FUNCTION_BLOCK FB_StatePMPSLimits_Test EXTENDS MotorTestSuite
(*
    Tests for FB_StatePMPSLimits

    This function block ensures that:
    - When not at our goal state, we cannot move away from our goal state
    - When at our goal state, we must stay within the state bounds
    - When at our goal state, we still obey other constraints like limit switches
*)
VAR
    stMotionStage: ST_MotionStage;
    fbMotionStage: FB_MotionStage;
    astPositionState: ARRAY[1..GeneralConstants.MAX_STATES] OF ST_PositionState;
    fbInternal1: FB_PositionStateInternal;
    fbInternal2: FB_PositionStateInternal;
    nInvalidState: UINT := 2;
    nGoalState: UINT := 4;
    nNotUpdatedState: UINT := 6;

    bInit: BOOL;
    nTestCounter: UINT;
    bOneTestDone: BOOL;
    fTestStartPos: LREAL;
    tonTimer: TON;
    bStatesReady: BOOL;
END_VAR


astPositionState[nGoalState].fPosition := 10;
astPositionState[nGoalState].fDelta := 1;
SetGoodState(astPositionState[nGoalState]);
astPositionState[nInvalidState].fPosition := 20;
astPositionState[nInvalidState].fDelta := 1;
astPositionState[nNotUpdatedState].fPosition := 20;
astPositionState[nNotUpdatedState].fDelta := 1;
SetGoodState(astPositionState[nNotUpdatedState]);
fbInternal1(
    stMotionStage:=stMotionStage,
    stPositionState:=astPositionState[nGoalState],
);
fbInternal2(
    stMotionStage:=stMotionStage,
    stPositionState:=astPositionState[nInvalidState],
);
fbMotionStage(stMotionStage:=stMotionStage);
bStatesReady:=astPositionState[nGoalState].bUpdated AND astPositionState[nInvalidState].bUpdated;

IF bStatesReady AND nTestCounter = 0 THEN
    // Don't run any tests until the states are ready
    nTestCounter := 1;
END_IF

TestInvalid(1);
TestNotUpdated(2);
TestBelow(3);
TestAbove(4);
TestAt(5);
TestDisabled(6);
TestLimits(7);

IF bOneTestDone THEN
    bOneTestDone := FALSE;
    nTestCounter := nTestCounter + 1;
    tonTimer(IN:=FALSE);
END_IF
// Use this timer to time out any tests that stall
tonTimer(
    IN:=bStatesReady,
    PT:=T#5s,
);

METHOD TestAbove
VAR_INPUT
    nTestID: UINT;
END_VAR
VAR_INST
    fbStateLimits: FB_StatePMPSLimits;
    fbFFHWO: FB_HardwareFFOutput := (bAutoReset := TRUE);
    fbMove: FB_TestHelperSetAndMove;

    bInit: BOOL;
END_VAR

TEST('TestAbove');
IF nTestCounter <> nTestID THEN
    RETURN;
END_IF

SetEnablesPMPS(stMotionStage);

// Set position to be above the goal's range
fbMove(
    stMotionStage:=stMotionStage,
    bExecute:=bInit,
    fStartPosition:=astPositionState[nGoalState].fPosition + 100 * astPositionState[nGoalState].fDelta,
    fGoalPosition:=astPositionState[nGoalState].fPosition + 100 * astPositionState[nGoalState].fDelta,
    fVelocity:=1,
    bHWEnable:=FALSE,
);
bInit := TRUE;
// Run our FB
fbStateLimits(
    stMotionStage:=stMotionStage,
    astPositionState:=astPositionState,
    fbFFHWO:=fbFFHWO,
    bEnable:=TRUE,
    nGoalStateIndex:=nGoalState,
);
fbFFHWO.EvaluateOutput();
// If we've set the position OR ran out of time to set the position, check the asserts
IF tonTimer.Q OR fbMove.bSetDone THEN
    AssertFalse(
        tonTimer.Q,
        'Timeout in test',
    );
    AssertEquals_LREAL(
        Expected:=fbMove.fStartPosition,
        Actual:=fbMove.fActPosition,
        Delta:=0.0001,
        Message:='Position was not set correctly',
    );
    AssertTrue(
        fbFFHWO.q_xFastFaultOut,
        'Fast fault in normal situation',
    );
    AssertFalse(
        fbStateLimits.bForwardEnabled,
        'Forward enabled when above goal',
    );
    AssertTrue(
        fbStateLimits.bBackwardEnabled,
        'Backward disabled when above goal',
    );
    bOneTestDone := TRUE;
    TEST_FINISHED();
END_IF
END_METHOD

METHOD TestAt
VAR_INPUT
    nTestID: UINT;
END_VAR
VAR_INST
    fbStateLimits: FB_StatePMPSLimits;
    fbFFHWO: FB_HardwareFFOutput := (bAutoReset := TRUE);
    fbMove: FB_TestHelperSetAndMove;

    bInit: BOOL;
END_VAR

TEST('TestAt');
IF nTestCounter <> nTestID THEN
    RETURN;
END_IF

SetEnablesPMPS(stMotionStage);

// Set position to be at the goal state
fbMove(
    stMotionStage:=stMotionStage,
    bExecute:=bInit,
    fStartPosition:=astPositionState[nGoalState].fPosition,
    fGoalPosition:=astPositionState[nGoalState].fPosition,
    fVelocity:=1,
    bHWEnable:=FALSE,
);
bInit := TRUE;
// Run our FB
fbStateLimits(
    stMotionStage:=stMotionStage,
    astPositionState:=astPositionState,
    fbFFHWO:=fbFFHWO,
    bEnable:=TRUE,
    nGoalStateIndex:=nGoalState,
);
fbFFHWO.EvaluateOutput();
// If we've set the position OR ran out of time to set the position, check the asserts
IF tonTimer.Q OR fbMove.bSetDone THEN
    AssertFalse(
        tonTimer.Q,
        'Timeout in test',
    );
    AssertEquals_LREAL(
        Expected:=fbMove.fStartPosition,
        Actual:=fbMove.fActPosition,
        Delta:=0.0001,
        Message:='Position was not set correctly',
    );
    AssertTrue(
        fbFFHWO.q_xFastFaultOut,
        'Fast fault in normal situation',
    );
    AssertTrue(
        fbStateLimits.bForwardEnabled,
        'Forward disabled when at goal',
    );
    AssertTrue(
        fbStateLimits.bBackwardEnabled,
        'Backward disabled when at goal',
    );
    bOneTestDone := TRUE;
    TEST_FINISHED();
END_IF
END_METHOD

METHOD TestBelow
VAR_INPUT
    nTestID: UINT;
END_VAR
VAR_INST
    fbStateLimits: FB_StatePMPSLimits;
    fbFFHWO: FB_HardwareFFOutput := (bAutoReset := TRUE);
    fbMove: FB_TestHelperSetAndMove;

    bInit: BOOL;
END_VAR

TEST('TestBelow');
IF nTestCounter <> nTestID THEN
    RETURN;
END_IF

SetEnablesPMPS(stMotionStage);

// Set position to be below the goal's range
fbMove(
    stMotionStage:=stMotionStage,
    bExecute:=bInit,
    fStartPosition:=astPositionState[nGoalState].fPosition - 100 * astPositionState[nGoalState].fDelta,
    fGoalPosition:=astPositionState[nGoalState].fPosition - 100 * astPositionState[nGoalState].fDelta,
    fVelocity:=1,
    bHWEnable:=FALSE,
);
bInit := TRUE;
// Run our FB
fbStateLimits(
    stMotionStage:=stMotionStage,
    astPositionState:=astPositionState,
    fbFFHWO:=fbFFHWO,
    bEnable:=bInit,
    nGoalStateIndex:=nGoalState,
);

fbFFHWO.EvaluateOutput();
// If we've set the position OR ran out of time to set the position, check the asserts
IF tonTimer.Q OR fbMove.bSetDone THEN
    AssertFalse(
        tonTimer.Q,
        'Timeout in test',
    );
    AssertEquals_LREAL(
        Expected:=fbMove.fStartPosition,
        Actual:=fbMove.fActPosition,
        Delta:=0.0001,
        Message:='Position was not set correctly',
    );
    AssertTrue(
        fbFFHWO.q_xFastFaultOut,
        'Fast fault in normal situation',
    );
    AssertFalse(
        fbStateLimits.bBackwardEnabled,
        'Backward enabled when below goal',
    );
    AssertTrue(
        fbStateLimits.bForwardEnabled,
        'Forward disabled when below goal',
    );
    bOneTestDone := TRUE;
    TEST_FINISHED();
END_IF
END_METHOD

METHOD TestDisabled
VAR_INPUT
    nTestID: UINT;
END_VAR
VAR_INST
    fbStateLimits: FB_StatePMPSLimits;
    fbFFHWO: FB_HardwareFFOutput := (bAutoReset := TRUE);
    fbMove: FB_TestHelperSetAndMove;

    bInit: BOOL;
END_VAR

TEST('TestDisabled');
IF nTestCounter <> nTestID THEN
    RETURN;
END_IF

SetEnablesPMPS(stMotionStage);

// Set position to be below the goal's range
fbMove(
    stMotionStage:=stMotionStage,
    bExecute:=bInit,
    fStartPosition:=astPositionState[nGoalState].fPosition - 100 * astPositionState[nGoalState].fDelta,
    fGoalPosition:=astPositionState[nGoalState].fPosition - 100 * astPositionState[nGoalState].fDelta,
    fVelocity:=1,
    bHWEnable:=FALSE,
);
bInit := TRUE;
// Run our FB
fbStateLimits(
    stMotionStage:=stMotionStage,
    astPositionState:=astPositionState,
    fbFFHWO:=fbFFHWO,
    bEnable:=FALSE,
    nGoalStateIndex:=nGoalState,
);

fbFFHWO.EvaluateOutput();
// If we've set the position OR ran out of time to set the position, check the asserts
IF tonTimer.Q OR fbMove.bSetDone THEN
    AssertFalse(
        tonTimer.Q,
        'Timeout in test',
    );
    AssertEquals_LREAL(
        Expected:=fbMove.fStartPosition,
        Actual:=fbMove.fActPosition,
        Delta:=0.0001,
        Message:='Position was not set correctly',
    );
    AssertTrue(
        fbFFHWO.q_xFastFaultOut,
        'Fast fault in normal situation',
    );
    AssertTrue(
        fbStateLimits.bBackwardEnabled,
        'Backward disabled when fb is supposed to be disabled',
    );
    AssertTrue(
        fbStateLimits.bForwardEnabled,
        'Forward disabled when fb is supposed to be disabled',
    );
    bOneTestDone := TRUE;
    TEST_FINISHED();
END_IF
END_METHOD

METHOD TestInvalid
VAR_INPUT
    nTestID: UINT;
END_VAR
VAR_INST
    fbStateLimits: FB_StatePMPSLimits;
    fbFFHWO: FB_HardwareFFOutput := (bAutoReset := TRUE);
END_VAR

TEST('TestInvalid');
IF nTestCounter <> nTestID THEN
    RETURN;
END_IF

SetEnablesPMPS(stMotionStage);

fbFFHWO.EvaluateOutput();
AssertTrue(
    fbFFHWO.q_xFastFaultOut,
    'Faulted prior to test',
);
// The invalid state should give us a fault
fbStateLimits(
    stMotionStage:=stMotionStage,
    astPositionState:=astPositionState,
    fbFFHWO:=fbFFHWO,
    bEnable:=TRUE,
    nGoalStateIndex:=nInvalidState,
);
fbFFHWO.EvaluateOutput();
AssertFalse(
    fbFFHWO.q_xFastFaultOut,
    'Invalid state did not fault',
);

bOneTestDone := TRUE;
TEST_FINISHED();
END_METHOD

METHOD TestLimits
VAR_INPUT
    nTestID: UINT;
END_VAR
VAR_INST
    fbStateLimits: FB_StatePMPSLimits;
    fbFFHWO: FB_HardwareFFOutput := (bAutoReset := TRUE);
    fbMove: FB_TestHelperSetAndMove;

    bInit: BOOL;
END_VAR

TEST('TestLimits');
IF nTestCounter <> nTestID THEN
    RETURN;
END_IF

SetEnablesPMPS(stMotionStage);
// Kill the limit switches for this test
stMotionStage.bLimitForwardEnable := FALSE;
stMotionStage.bLimitBackwardEnable := FALSE;

// Set position to be at the goal state
fbMove(
    stMotionStage:=stMotionStage,
    bExecute:=bInit,
    fStartPosition:=astPositionState[nGoalState].fPosition,
    fGoalPosition:=astPositionState[nGoalState].fPosition,
    fVelocity:=1,
    bHWEnable:=FALSE,
);
bInit := TRUE;

// Run our FB
fbStateLimits(
    stMotionStage:=stMotionStage,
    astPositionState:=astPositionState,
    fbFFHWO:=fbFFHWO,
    bEnable:=TRUE,
    nGoalStateIndex:=nGoalState,
);
fbFFHWO.EvaluateOutput();
// If we've set the position OR ran out of time to set the position, check the asserts
IF tonTimer.Q OR fbMove.bSetDone THEN
    AssertFalse(
        tonTimer.Q,
        'Timeout in test',
    );
    AssertEquals_LREAL(
        Expected:=fbMove.fStartPosition,
        Actual:=fbMove.fActPosition,
        Delta:=0.0001,
        Message:='Position was not set correctly',
    );
    AssertTrue(
        fbFFHWO.q_xFastFaultOut,
        'Fast fault in normal situation',
    );
    AssertFalse(
        fbStateLimits.bForwardEnabled,
        'Forward enabled with limit hit',
    );
    AssertFalse(
        fbStateLimits.bBackwardEnabled,
        'Backward enabled with limit hit',
    );
    bOneTestDone := TRUE;
    TEST_FINISHED();
END_IF
END_METHOD

METHOD TestNotUpdated
VAR_INPUT
    nTestID: UINT;
END_VAR
VAR_INST
    fbStateLimits: FB_StatePMPSLimits;
    fbFFHWO: FB_HardwareFFOutput := (bAutoReset := TRUE);
END_VAR

TEST('TestNotUpdated');
IF nTestCounter <> nTestID THEN
    RETURN;
END_IF

SetEnablesPMPS(stMotionStage);

fbFFHWO.EvaluateOutput();
AssertTrue(
    fbFFHWO.q_xFastFaultOut,
    'Faulted prior to test',
);
// The invalid state should give us a fault
fbStateLimits(
    stMotionStage:=stMotionStage,
    astPositionState:=astPositionState,
    fbFFHWO:=fbFFHWO,
    bEnable:=TRUE,
    nGoalStateIndex:=nNotUpdatedState,
);
fbFFHWO.EvaluateOutput();
AssertFalse(
    fbFFHWO.q_xFastFaultOut,
    'Not updated state did not fault',
);

bOneTestDone := TRUE;
TEST_FINISHED();
END_METHOD

END_FUNCTION_BLOCK

(* stored: Version 1.1.0.1, ProductVersion 3.1.4022.18
   POU FB_StatePMPSLimits_Test: Id {5c47f34f-d68e-4ecd-b2fb-e45bba741378}, SpecialFunc None
   Method TestAbove: Id {bc286948-b217-49e2-8136-d78acdf6793d}
   Method TestAt: Id {eeabf203-9322-4bdb-a96d-693569eb0c9f}
   Method TestBelow: Id {98c46d12-8b7c-43dd-b3b3-9f3e17c240da}
   Method TestDisabled: Id {c7db8114-667b-44b5-9eaa-1b1048940e05}
   Method TestInvalid: Id {af1a625f-1614-486f-ac30-8390914f582a}
   Method TestLimits: Id {6546d47a-b549-4011-b1e7-32f110cda4b9}
   Method TestNotUpdated: Id {e3e62099-da37-4d9e-b58b-650fd1e6c70e} *)
